// TIA Portal V18 export
FUNCTION "AHUExtractDumperctCtrl" : Void   // FC60307, LAD
{ S7_Optimized_Access := 'TRUE' }
VERSION : 0.1
// stored: AutoNumber false, IsIECCheckEnabled false, SetENOAutomatically false, UDAEnableTagReadback false
BEGIN
END_FUNCTION
